// TwinCAT 3 PLC project PLC
// ProgramVersion: 3.1.4023.0
// libraries:
//   EfficientIO Communicator, * (EfficientIO)
//   Lynus Energy Basic, * (Lynus AG)
//   Lynus Energy ModbusRTU, * (Lynus AG)
//   Lynus Energy ModbusTCP, * (Lynus AG)
//   Lynus Persistent Data V1, * (Lynus AG)
//   Lynus Sensor Basic, * (Lynus AG)
//   Lynus Standards, * (Lynus AG)
//   Tc2_ModbusSrv, * (Beckhoff Automation GmbH)
//   Tc2_Standard, * (Beckhoff Automation GmbH)
//   Tc2_System, * (Beckhoff Automation GmbH)
//   Tc2_Utilities, * (Beckhoff Automation GmbH)
//   Tc3_Module, * (Beckhoff Automation GmbH)
// project tree:
//   DUTs/ eByteOrder.TcDUT
//   / Fast_Task.TcTTO, Middle_Task.TcTTO, Slow_Task.TcTTO
//   FBs/ FB_CV_WORD_TO_DWORD.TcPOU, FB_EnergyCounter.TcPOU, FB_Honeywell_Excange_Data.TcPOU, FB_HouseC_Power_Virtual_v2.TcPOU
//   POUs/ prgComLynus.TcPOU, prgCS.TcPOU, prgEHE.TcPOU, prgEMS.TcPOU, prgGrid.TcPOU, prgHoneywell.TcPOU, prgHouse.TcPOU, prgKNX.TcPOU, prgPerData.TcPOU, prgPV.TcPOU, prgRWLynus.TcPOU, prgVarLynus.TcPOU, prgXelect.TcPOU
// real-time tasks:
//   TASK Fast Task: cycle T#5ms, priority 6, ADS port 351
//   TASK Middle Task: cycle T#10ms, priority 8, ADS port 352
//   TASK Slow Task: cycle T#20ms, priority 10, ADS port 353
// I/O:
//   DEVICE Gerät 2 (CX-BK)
//     Box 1 (CX-BK)
// variable links:
//   PLC/PLC Instance <-> Device 2 (CX-BK)/Box 1 (CX-BK)
//     Fast_Task Inputs/prgCS.fbRTUMaster.fbmodbusmaster.InData/D[{0..21}] <-> Term 4 (KL6041)/Channel 1/Data In {0..21}  (22 links)
//     Fast_Task Inputs/prgCS.fbRTUMaster.fbmodbusmaster.InData/Status <-> Term 4 (KL6041)/Channel 1/Status
//     Fast_Task Inputs/prgKNX.fbKBusState.uiKBusState_OUT <-> Inputs/State
//     Fast_Task Outputs/prgCS.fbRTUMaster.fbmodbusmaster.OutData/Ctrl <-> Term 4 (KL6041)/Channel 1/Ctrl
//     Fast_Task Outputs/prgCS.fbRTUMaster.fbmodbusmaster.OutData/D[{0..21}] <-> Term 4 (KL6041)/Channel 1/Data Out {0..21}  (22 links)
//     Middle_Task Inputs/prgEHE.fbH08_1.fbAOEHE.usiState <-> Term 2 (KL4404)/Channel 1/Status
//     Middle_Task Inputs/prgEHE.fbH08_2.fbAOEHE.usiState <-> Term 2 (KL4404)/Channel 2/Status
//     Middle_Task Inputs/prgEHE.fbH09_1.fbAOEHE.usiState <-> Term 2 (KL4404)/Channel 3/Status
//     Middle_Task Inputs/prgKNX.fbKNXMaster.arrKNXKL6301ComIn @bit {16..184 step 8} <-> Term 3 (KL6301)/Channel 1/Input Data {1..22}  (22 links)
//     Middle_Task Inputs/prgKNX.fbKNXMaster.arrKNXKL6301ComIn <-> Term 3 (KL6301)/Channel 1/Parameter Status
//     Middle_Task Outputs/prgEHE.fbH08_1.fbAOEHE.iDataOut <-> Term 2 (KL4404)/Channel 1/Daten Aus
//     Middle_Task Outputs/prgEHE.fbH08_2.fbAOEHE.iDataOut <-> Term 2 (KL4404)/Channel 2/Daten Aus
//     Middle_Task Outputs/prgEHE.fbH09_1.fbAOEHE.iDataOut <-> Term 2 (KL4404)/Channel 3/Daten Aus
//     Middle_Task Outputs/prgKNX.fbKNXMaster.arrKNXKL6301ComOut @bit {16..184 step 8} <-> Term 3 (KL6301)/Channel 1/Output Data {1..22}  (22 links)
//     Middle_Task Outputs/prgKNX.fbKNXMaster.arrKNXKL6301ComOut <-> Term 3 (KL6301)/Channel 1/Parameter Control

CONFIGURATION PLC
    RESOURCE PLC ON TwinCAT3
        TASK Fast_Task(INTERVAL := T#5ms, PRIORITY := 6);
        TASK Middle_Task(INTERVAL := T#10ms, PRIORITY := 8);
        TASK Slow_Task(INTERVAL := T#20ms, PRIORITY := 10);
        PROGRAM prgRWLynus WITH Fast_Task : prgRWLynus;
        PROGRAM prgVarLynus WITH Fast_Task : prgVarLynus;
        PROGRAM prgCS WITH Fast_Task : prgCS;
        PROGRAM prgEHE WITH Middle_Task : prgEHE;
        PROGRAM prgEMS WITH Middle_Task : prgEMS;
        PROGRAM prgHoneywell WITH Middle_Task : prgHoneywell;
        PROGRAM prgKNX WITH Middle_Task : prgKNX;
        PROGRAM prgPV WITH Middle_Task : prgPV;
        PROGRAM prgXelect WITH Middle_Task : prgXelect;
        PROGRAM prgPerData WITH Middle_Task : prgPerData;
        PROGRAM prgHouse WITH Middle_Task : prgHouse;
        PROGRAM prgGrid WITH Middle_Task : prgGrid;
        PROGRAM prgComLynus WITH Slow_Task : prgComLynus;
    END_RESOURCE
END_CONFIGURATION

// ---- DUTs/eByteOrder.TcDUT
TYPE eByteOrder :
(
	eBigEndian	:= 0,
	eLittleEndian	:= 1
);
END_TYPE

// ---- POUs/prgRWLynus.TcPOU
PROGRAM prgRWLynus
VAR
	fbRW1		: FB_ReadWrite;
	fbRW2		: FB_ReadWrite;
	fbRW3		: FB_ReadWrite;
	fbRW4		: FB_ReadWrite;
	fbRW5		: FB_ReadWrite;
	fbRW6		: FB_ReadWrite;
END_VAR

fbRW1();
fbRW2();
fbRW3();
fbRW4();
fbRW5();
fbRW6();

END_PROGRAM

// ---- POUs/prgVarLynus.TcPOU
PROGRAM prgVarLynus
VAR
	fbVar			: FB_VarInfo;
END_VAR

fbVar(
	bReadInfo:= , 
	eTMCFile:= eSelectTMCFile.eUseTMCFile, 
	eSavePositionTMCFile:= eSavePositionOnPLC.ePostionHardDisk, 
	udiCounterFoundVariables=> , 
	bError=> , 
	bBusy=> , 
	byProgress=> , 
	udiErrorCodeOut=> , 
	eErrorVarInfo_Out=> , 
	sVarWithError=> );

END_PROGRAM

// ---- POUs/prgCS.TcPOU
PROGRAM prgCS
VAR
	fbRTUMaster					: FB_KL6xxx_ModbusRTU_22B_Master;
	byErrorwarningRTU			: BYTE;									//{#lynus.ag#()}
	fbCS1						: FB_ECS_Schrack_EM_CionHome;			//{#lynus.ag#()}
	fbCS2						: FB_ECS_Schrack_EM_CionHome;			//{#lynus.ag#()}
	fbCS3						: FB_ECS_Schrack_EM_CionHome;			//{#lynus.ag#()}
	bCarConnCS1					: BOOL;									//{#lynus.ag#()}
	bCarConnCS2					: BOOL;									//{#lynus.ag#()}
	bCarConnCS3					: BOOL;									//{#lynus.ag#()}
	bOnEmergPowerOffCS1			: BOOL;									//{#lynus.ag#()}
	bOnEmergPowerOffCS2			: BOOL;									//{#lynus.ag#()}
	bOnEmergPowerOffCS3			: BOOL;									//{#lynus.ag#()}
	bSOnEmergPowerOffCS1		: BOOL;									//{#lynus.ag#()}
	bSOnEmergPowerOffCS2		: BOOL;									//{#lynus.ag#()}
	bSOnEmergPowerOffCS3		: BOOL;									//{#lynus.ag#()}
	byErrorWarningCS1			: BYTE;									//{#lynus.ag#()}
	byErrorWarningCS2			: BYTE;									//{#lynus.ag#()}
	byErrorWarningCS3			: BYTE;									//{#lynus.ag#()}
	wCPStateCS1					: WORD;									//{#lynus.ag#()}
	bChargingReleaseInavlidCS1	: BOOL;									//{#lynus.ag#()}
	rChargingTimeInMinCS1		: REAL;									//{#lynus.ag#()}
	wCPStateCS2					: WORD;									//{#lynus.ag#()}
	bChargingReleaseInavlidCS2	: BOOL;									//{#lynus.ag#()}
	rChargingTimeInMinCS2		: REAL;									//{#lynus.ag#()}
	wCPStateCS3					: WORD;									//{#lynus.ag#()}
	bChargingReleaseInavlidCS3	: BOOL;									//{#lynus.ag#()}
	rChargingTimeInMinCS3		: REAL;									//{#lynus.ag#()}
	byErrorCounter				: BYTE;									//{#lynus.ag#()}
	FpErrror					: R_TRIG;
END_VAR

//Power Data
//Each CS has 14kW

fbRTUMaster(
	bConfigTerminal:= , 
	uiKBusState_IN:= prgKNX.fbKBusState.uiKBusState_OUT, 
	bBusy=> , 
	byErrorWarning=> , 
	byActualAdressInUse=> , 
	diNrOfMBRTUMasterLine_OUT=> , 
	eMessageMBRTUMaster=> , 
	bTerminalIsConfigured=> );

fbRTUMaster(
	bConfigTerminal:= , 
	bBusy=> , 
	byErrorWarning=> , 
	diNrOfMBRTUMasterLine_OUT=> , 
	eMessageMBRTUMaster=> , 
	bTerminalIsConfigured=> );

byErrorwarningRTU := fbRTUMaster.byErrorWarning;

FpErrror(CLK:= byErrorwarningRTU = 2, Q=> );
	IF FpErrror.Q THEN byErrorCounter := byErrorCounter + 1; END_IF
	
//Garage 1 near Door	
fbCS1.stSetupECS.bOnEmergPowerOff := bOnEmergPowerOffCS1;

fbCS1(
	bEnable:= , 
	bPowerDataInvers:= , 
	byMBAdress:= 1, 
	diNrOfMBRTUMasterLine_IN:= fbRTUMaster.diNrOfMBRTUMasterLine_OUT, 
	diNrOfEMS_IN:= prgEMS.EMS.diNrOfEMS_OUT, 
	diNrOfEM_IN_CS:= , 
	stSetupECS:= , 
	stDataECS=> , 
	eSchrackErrors=> , 
	diNrOfECS_OUT=> );

wCPStateCS1:= fbCS1.wCPStateECS;
	bChargingReleaseInavlidCS1 := fbCS1.bChargingReleaseInavlid;
		rChargingTimeInMinCS1 := fbCS1.stDataECS.arrChargingTimeInMin[1];
			byErrorWarningCS1 := fbCS1.stDataECS.byErrorWarning;
				bCarConnCS1 := fbCS1.stDataECS.bCarConnected;
					bSOnEmergPowerOffCS1 := fbCS1.stDataECS.bSOnEmergPowerOff;
	
//Between CS1	
fbCS2.stSetupECS.bOnEmergPowerOff := bOnEmergPowerOffCS2;

fbCS2(
	bEnable:= , 
	bPowerDataInvers:= , 
	byMBAdress:= 2, 
	diNrOfMBRTUMasterLine_IN:= fbRTUMaster.diNrOfMBRTUMasterLine_OUT, 
	diNrOfEMS_IN:= prgEMS.EMS.diNrOfEMS_OUT, 
	diNrOfEM_IN_CS:= , 
	stSetupECS:= , 
	stDataECS=> , 
	eSchrackErrors=> , 
	diNrOfECS_OUT=> );

wCPStateCS2:= fbCS2.wCPStateECS;
	bChargingReleaseInavlidCS2 := fbCS2.bChargingReleaseInavlid;
		rChargingTimeInMinCS2 := fbCS2.stDataECS.arrChargingTimeInMin[1];
			byErrorWarningCS2 := fbCS2.stDataECS.byErrorWarning;
				bCarConnCS2 := fbCS2.stDataECS.bCarConnected;
					bSOnEmergPowerOffCS2 := fbCS2.stDataECS.bSOnEmergPowerOff;	
	
//Outdoor CS
fbCS3.stSetupECS.bOnEmergPowerOff := bOnEmergPowerOffCS3;

fbCS3(
	bEnable:= , 
	bPowerDataInvers:= , 
	byMBAdress:= 3, 
	diNrOfMBRTUMasterLine_IN:= fbRTUMaster.diNrOfMBRTUMasterLine_OUT, 
	diNrOfEMS_IN:= prgEMS.EMS.diNrOfEMS_OUT, 
	diNrOfEM_IN_CS:= , 
	stSetupECS:= , 
	stDataECS=> , 
	eSchrackErrors=> , 
	diNrOfECS_OUT=> );
	
wCPStateCS3:= fbCS3.wCPStateECS;
	bChargingReleaseInavlidCS3 := fbCS3.bChargingReleaseInavlid;
		rChargingTimeInMinCS3 := fbCS3.stDataECS.arrChargingTimeInMin[1];
			byErrorWarningCS3 := fbCS3.stDataECS.byErrorWarning;
				bCarConnCS3 := fbCS3.stDataECS.bCarConnected;
					bSOnEmergPowerOffCS3 := fbCS3.stDataECS.bSOnEmergPowerOff;

END_PROGRAM

// ---- POUs/prgKNX.TcPOU
PROGRAM prgKNX
VAR
	fbKBusState				: FB_K_Bus_State;
	fbKNXMaster				: FB_KL6301_KNX_Master;
	fbRampHeating			: FB_OBC_OnOff_KNX;				//{#lynus.ag#()}
	fbTreeHeating			: FB_OBC_OnOff_KNX;				//{#lynus.ag#()}
	fbPumpFishSea			: FB_OBC_OnOff_KNX;				//{#lynus.ag#()}
	fbPumpSwimSea			: FB_OBC_OnOff_KNX;				//{#lynus.ag#()}
	bOnEmergPowerOffRH		: BOOL;							//{#lynus.ag#()}
	bOnEmergPowerOffTH		: BOOL;							//{#lynus.ag#()}
	bOnEmergPowerOffPFish	: BOOL;							//{#lynus.ag#()}
	bOnEmergPowerOffPSwim	: BOOL;							//{#lynus.ag#()}
	bSOnEmergPowerOffRH		: BOOL;							//{#lynus.ag#()}
	bSOnEmergPowerOffTH		: BOOL;							//{#lynus.ag#()}
	bSOnEmergPowerOffPFish	: BOOL;							//{#lynus.ag#()}
	bSOnEmergPowerOffPSwim	: BOOL;							//{#lynus.ag#()}
	byErrorWarningRH		: BYTE;							//{#lynus.ag#()}
	byErrorWarningTH		: BYTE;							//{#lynus.ag#()}
	byErrorWarningPFish		: BYTE;							//{#lynus.ag#()}
	byErrorWarningPSwim		: BYTE;							//{#lynus.ag#()}
END_VAR

//Power Data
//Ramp Heating 34kw
//Three Heating 13kW 
//Fish Sea pump 7.5kW
//Swim Sea Pump 7.5kw

//K-Bus State
fbKBusState(uiKBusState_OUT=> );

//Configure the KXN Master
fbKNXMaster.stPhysAddrTerminal.Area := 1;
	fbKNXMaster.stPhysAddrTerminal.Device := 160;
		fbKNXMaster.stPhysAddrTerminal.Line := 9;
		
fbKNXMaster.arrGroupFilter[1].GROUP_ADDR.MAIN := 6;
	fbKNXMaster.arrGroupFilter[1].GROUP_ADDR.NUMBER := 0;
		fbKNXMaster.arrGroupFilter[1].GROUP_ADDR.SUB_MAIN := 1;
fbKNXMaster.arrGroupFilter[1].GROUP_LEN := 4;	
	
fbKNXMaster(
	stPhysAddrTerminal:= , 
	arrGroupFilter:= , 
	iKL6301Mode:= 0, 
	uiKBusState_IN:= fbKBusState.uiKBusState_OUT, 
	bActive=> , 
	bReady=> , 
	byErrorWarning=> , 
	diNrOfKNXMasterLine_OUT=> , 
	eMessageKNXMaster=> );

fbTreeHeating.strGroupAddr.MAIN := 6;
	fbTreeHeating.strGroupAddr.SUB_MAIN := 1;
		fbTreeHeating.strGroupAddr.NUMBER := 0;	

fbTreeHeating.stSetupOBC.bOnEmergPowerOff := bOnEmergPowerOffTH;
	
fbTreeHeating(
	bEnable:= , 
	bPowerDataInvers:= , 
	diNrOfKNXMasterLine_IN:= fbKNXMaster.diNrOfKNXMasterLine_OUT, 
	diNrOfEMS_IN:= prgEMS.EMS.diNrOfEMS_OUT, 
	diNrOfEM_IN_OBC:= , 
	stSetupOBC:= , 
	strGroupAddr:= , 
	stDataOBC=> , 
	diNrOfOBC_OUT=> );

byErrorWarningTH := fbTreeHeating.stDataOBC.byErrorWarning;	
	bSOnEmergPowerOffTH := fbTreeHeating.stDataOBC.bSOnEmergPowerOff;	
	
fbPumpFishSea.strGroupAddr.MAIN := 6;
	fbPumpFishSea.strGroupAddr.SUB_MAIN := 1;
		fbPumpFishSea.strGroupAddr.NUMBER := 2;	

fbPumpFishSea.stSetupOBC.bOnEmergPowerOff := bOnEmergPowerOffPFish;
	
fbPumpFishSea(
	bEnable:= , 
	bPowerDataInvers:= , 
	diNrOfKNXMasterLine_IN:= fbKNXMaster.diNrOfKNXMasterLine_OUT, 
	diNrOfEMS_IN:= prgEMS.EMS.diNrOfEMS_OUT, 
	diNrOfEM_IN_OBC:= , 
	stSetupOBC:= , 
	strGroupAddr:= , 
	stDataOBC=> , 
	diNrOfOBC_OUT=> );

byErrorWarningPFish := fbPumpFishSea.stDataOBC.byErrorWarning;
	bSOnEmergPowerOffPFish := fbPumpFishSea.stDataOBC.bSOnEmergPowerOff;		
	
fbPumpSwimSea.strGroupAddr.MAIN := 6;
	fbPumpSwimSea.strGroupAddr.SUB_MAIN := 1;
		fbPumpSwimSea.strGroupAddr.NUMBER := 3;	

fbPumpSwimSea.stSetupOBC.bOnEmergPowerOff := bOnEmergPowerOffPSwim;
	
fbPumpSwimSea(
	bEnable:= , 
	bPowerDataInvers:= , 
	diNrOfKNXMasterLine_IN:= fbKNXMaster.diNrOfKNXMasterLine_OUT, 
	diNrOfEMS_IN:= prgEMS.EMS.diNrOfEMS_OUT, 
	diNrOfEM_IN_OBC:= , 
	stSetupOBC:= , 
	strGroupAddr:= , 
	stDataOBC=> , 
	diNrOfOBC_OUT=> );

byErrorWarningPSwim := fbPumpSwimSea.stDataOBC.byErrorWarning;	
	bSOnEmergPowerOffPSwim := fbPumpSwimSea.stDataOBC.bSOnEmergPowerOff;
	
fbRampHeating.strGroupAddr.MAIN := 6;
	fbRampHeating.strGroupAddr.SUB_MAIN := 1;
		fbRampHeating.strGroupAddr.NUMBER := 1;	

fbRampHeating.stSetupOBC.bOnEmergPowerOff := bOnEmergPowerOffRH;
	
fbRampHeating(
	bEnable:= , 
	bPowerDataInvers:= , 
	diNrOfKNXMasterLine_IN:= fbKNXMaster.diNrOfKNXMasterLine_OUT, 
	diNrOfEMS_IN:= prgEMS.EMS.diNrOfEMS_OUT, 
	diNrOfEM_IN_OBC:= , 
	stSetupOBC:= , 
	strGroupAddr:= , 
	stDataOBC=> , 
	diNrOfOBC_OUT=> );
	
byErrorWarningRH := fbRampHeating.stDataOBC.byErrorWarning;	
	bSOnEmergPowerOffRH := fbRampHeating.stDataOBC.bSOnEmergPowerOff;

END_PROGRAM

// ---- POUs/prgEMS.TcPOU
PROGRAM prgEMS
VAR
	EMS					: FB_EMS;			//{#lynus.ag#()}
	iMassageEMS			: INT;				//{#lynus.ag#()}
	fbreboot			: NT_Reboot;
END_VAR

EMS(
	bEnable:= , 
	diNrOfEM_IN_ECS:= , 
	stSetupEMS:= , 
	eOperationMode:= ,
	eSpeedModeBackendController:= E_SpeedModeBackendController_EMS.eSlow, 
	eSpeedModeLocalController:= E_SpeedModeLocalController_EMS.eBalanced,
	eMessageEMS=> , 
	bStateEnable=> , 
	bStateAllowChrgFromGrid=> , 
	bMissingPowerData=> , 
	bSurplusAvailable=> , 
	bActivateHP=> , 
	bControllingState=> , 
	byProgress=> , 
	diNrOfEMS_OUT=> , 
	rHeartbeat=> , 
	rErrorWarning=> , 
	rEnergyOptReady=> , 
	rNewBattPower=> , 
	arrMinPrioReached=> , 
	arrMaxPrioReached=> );
	
iMassageEMS := ems.eMessageEMS;

fbreboot(
	NETID:= , 
	DELAY:= , 
	START:= , 
	TMOUT:= , 
	BUSY=> , 
	ERR=> , 
	ERRID=> );

END_PROGRAM

// ---- POUs/prgEHE.TcPOU
PROGRAM prgEHE
VAR
	fbTempH08					: FB_TempS_Ext_Input;
	fbTempH09					: FB_TempS_Ext_Input;
	fbH08_1						: FB_EHE_Linear_AO;			//{#lynus.ag#()}
	fbH08_2						: FB_EHE_Linear_AO;			//{#lynus.ag#()}
	fbH09_1						: FB_EHE_Linear_AO;			//{#lynus.ag#()}
	bSOnEmergPowerOffH08_1		: BOOL;						//{#lynus.ag#()}
	bSOnEmergPowerOffH08_2		: BOOL;						//{#lynus.ag#()}
	bSOnEmergPowerOffH09_1		: BOOL;						//{#lynus.ag#()}
	byErrorWarningH08_1			: BYTE;						//{#lynus.ag#()}
	byErrorWarningH08_2			: BYTE;						//{#lynus.ag#()}
	byErrorWarningH09_1			: BYTE;						//{#lynus.ag#()}
END_VAR
VAR PERSISTENT
	bOnEmergPowerOffH08_1		: BOOL;						//{#lynus.ag#()}
	bOnEmergPowerOffH08_2		: BOOL;						//{#lynus.ag#()}
	bOnEmergPowerOffH09_1		: BOOL;						//{#lynus.ag#()}
END_VAR

//Power Data
//each Heating Element 9kW

fbTempH08(
	bEnable:= TRUE, 
	rTemperatureOffset:= , 
	bExtErrorTemp:= prgHoneywell.fbHoneywellCntr.bErrorFunction OR prgHoneywell.fbHoneywellCntr.bErrorTemp_H08_Below OR prgHoneywell.fbHoneywellCntr.bErrorTemp_H08_Top, 
	rExtTempValue:= (prgHoneywell.fbHoneywellCntr.rBufferTemp_H08_Below + prgHoneywell.fbHoneywellCntr.rBufferTemp_H08_Top) / 2, 
	stDataTempS=> , 
	diNrOfTempS_OUT=> );
	
fbTempH09(
	bEnable:= TRUE, 
	rTemperatureOffset:= , 
	bExtErrorTemp:= prgHoneywell.fbHoneywellCntr.bErrorFunction OR prgHoneywell.fbHoneywellCntr.bErrorTemp_H09_WW, 
	rExtTempValue:= prgHoneywell.fbHoneywellCntr.rBufferTemp_H09_WW, 
	stDataTempS=> , 
	diNrOfTempS_OUT=> );

//Buffer House	
fbH08_1.stSetupEHE.bOnEmergPowerOff := bOnEmergPowerOffH08_1;
	fbH08_1.stSetupEHE.bDisableLegionellaPr := TRUE;
	
fbH08_1(
	bEnable:= , 
	bPowerDataInvers:= , 
	bNoLinear:= FALSE,
	diNrOfEMS_IN:= prgEMS.EMS.diNrOfEMS_OUT, 
	diNrOfEM_IN_EHE:= , 
	diNrOfTempS_IN:= fbTempH08.diNrOfTempS_OUT, 
	stSetupEHE:= , 
	stDataEHE=> , 
	diNrOfEHE_OUT=> , 
	rTargetPowerForExtFunc=> );	
	
byErrorWarningH08_1 := fbH08_1.stDataEHE.byErrorWarning;
	bSOnEmergPowerOffH08_1 := fbH08_1.stDataEHE.bSOnEmergPowerOff;

fbH08_2.stSetupEHE.bOnEmergPowerOff := bOnEmergPowerOffH08_2;
	fbH08_2.stSetupEHE.bDisableLegionellaPr := TRUE;
	
fbH08_2(
	bEnable:= , 
	bPowerDataInvers:= , 
	bNoLinear:= FALSE,
	diNrOfEMS_IN:= prgEMS.EMS.diNrOfEMS_OUT, 
	diNrOfEM_IN_EHE:= , 
	diNrOfTempS_IN:= fbTempH08.diNrOfTempS_OUT, 
	stSetupEHE:= , 
	stDataEHE=> , 
	diNrOfEHE_OUT=> , 
	rTargetPowerForExtFunc=> );

byErrorWarningH08_2 := fbH08_2.stDataEHE.byErrorWarning;
	bSOnEmergPowerOffH08_2 := fbH08_2.stDataEHE.bSOnEmergPowerOff;	
	
//Warmwater Boiler	
fbH09_1.stSetupEHE.bOnEmergPowerOff := bOnEmergPowerOffH09_1;

fbH09_1(
	bEnable:= , 
	bPowerDataInvers:= , 
	bNoLinear:= FALSE,
	diNrOfEMS_IN:= prgEMS.EMS.diNrOfEMS_OUT, 
	diNrOfEM_IN_EHE:= , 
	diNrOfTempS_IN:= fbTempH09.diNrOfTempS_OUT, 
	stSetupEHE:= , 
	stDataEHE=> , 
	diNrOfEHE_OUT=> , 
	rTargetPowerForExtFunc=> );
	
byErrorWarningH09_1 := fbH09_1.stDataEHE.byErrorWarning;
	bSOnEmergPowerOffH09_1 := fbH09_1.stDataEHE.bSOnEmergPowerOff;

END_PROGRAM

// ---- POUs/prgHoneywell.TcPOU
PROGRAM prgHoneywell
VAR
	fbHoneywellCntr			: FB_Honeywell_Excange_Data;
	fbTempH01				: FB_TempS_Ext_Input;
	fbH01_1					: FB_EHE_Linear_AO;			//{#lynus.ag#()}
	fbH01_2					: FB_EHE_Linear_AO;			//{#lynus.ag#()}
	fbH01_3					: FB_EHE_Linear_AO;			//{#lynus.ag#()}
	bSOnEmergPowerOffH01_1	: BOOL;						//{#lynus.ag#()}
	bSOnEmergPowerOffH01_2	: BOOL;						//{#lynus.ag#()}
	bSOnEmergPowerOffH01_3	: BOOL;						//{#lynus.ag#()}
	rBufferTemp_H01_Top		: REAL;						//{#lynus.ag#()}
	rBufferTemp_H01_Below	: REAL;						//{#lynus.ag#()}
	rBufferTemp_H08_Top		: REAL;						//{#lynus.ag#()}
	rBufferTemp_H08_Below	: REAL;						//{#lynus.ag#()}
	bErrorHoneywell			: BOOL;						//{#lynus.ag#()}
	byErrorWarningH01_1		: BYTE;						//{#lynus.ag#()}
	byErrorWarningH01_2		: BYTE;						//{#lynus.ag#()}
	byErrorWarningH01_3		: BYTE;						//{#lynus.ag#()}
	dwHeatingMeterHouse		: DWORD;					//{#lynus.ag#()}
	dwHeatingMeterStable	: DWORD;					//{#lynus.ag#()}
	dwWaterMeterMain1		: DWORD;					//{#lynus.ag#()}
	dwWaterMeterService1	: DWORD;					//{#lynus.ag#()}
	dwWaterMeterStable1		: DWORD;					//{#lynus.ag#()}
	dwElectricMeterCounter	: DWORD;					//{#lynus.ag#()}
	dwElectricMeterPower	: LREAL;					//{#lynus.ag#()}
END_VAR
VAR PERSISTENT
	bOnEmergPowerOffH01_1	: BOOL;						//{#lynus.ag#()}
	bOnEmergPowerOffH01_2	: BOOL;						//{#lynus.ag#()}
	bOnEmergPowerOffH01_3	: BOOL;						//{#lynus.ag#()}
END_VAR

//Creator : Kai Ebensperger
//Company : Lynus AG
//Updated : M.Schwarzmann
//Date : 11.07.2022
//Version : 1.0.0.4

//changes
//1.0.0.1 : added dwWaterMeterMain, dwWaterMeterService, dwElectricMeterCounter, dwElectricMeterPower at fbHoneywellCntr
//1.0.0.2 : changed Variable dwElectricMeterPower from Type REAL to LREAL
//1.0.0.3 : re-named Variables dwWaterMeterMain, dwWaterMeterService
//1.0.0.4 : added dwWaterMeterStable1


//Power Data
//Each EHE 9 kW

fbHoneywellCntr(
	bEnable:= TRUE, 
	byUnitID:= 1, 
	rTargetPowerEHEH01_1:= fbH01_1.rTargetPowerForExtFunc, 
	rTargetPowerEHEH01_2:= fbH01_2.rTargetPowerForExtFunc, 
	rTargetPowerEHEH01_3:= fbH01_3.rTargetPowerForExtFunc, 
	rTargetPowerEHEH08_1:= prgEHE.fbH08_1.rTargetPowerForExtFunc, 
	rTargetPowerEHEH08_2:= prgEHE.fbH08_2.rTargetPowerForExtFunc, 
	rTargetPowerEHEH09_1:= prgEHE.fbH09_1.rTargetPowerForExtFunc, 
	sIPAdress:= '10.68.10.60', 
	bErrorTemp_H01_Top=> , 
	bErrorTemp_H01_Below=> , 
	bErrorTemp_H08_Top=> , 
	bErrorTemp_H08_Below=> , 
	bErrorTemp_H09_WW=> , 
	bErrorFunction=> bErrorHoneywell, 
	dwHeatingMeterHouse=> dwHeatingMeterHouse,
	dwHeatingMeterStable=> dwHeatingMeterStable,
	dwWaterMeterMain1=> dwWaterMeterMain1,
	dwWaterMeterService1=> dwWaterMeterService1,
	dwWaterMeterStable1=> dwWaterMeterStable1,
	dwElectricMeterCounter=> dwElectricMeterCounter,
	dwElectricMeterPower=> dwElectricMeterPower,
	rBufferTemp_H01_Top=> rBufferTemp_H01_Top, 
	rBufferTemp_H01_Below=> rBufferTemp_H01_Below, 
	rBufferTemp_H08_Top=> rBufferTemp_H08_Top, 
	rBufferTemp_H08_Below=> rBufferTemp_H08_Below, 
	rBufferTemp_H09_WW=> );

fbTempH01(
	bEnable:= TRUE, 
	rTemperatureOffset:= , 
	bExtErrorTemp:= fbHoneywellCntr.bErrorFunction OR fbHoneywellCntr.bErrorTemp_H01_Below OR fbHoneywellCntr.bErrorTemp_H01_Top, 
	rExtTempValue:= (fbHoneywellCntr.rBufferTemp_H01_Below + fbHoneywellCntr.rBufferTemp_H01_Top) / 2, 
	stDataTempS=> , 
	diNrOfTempS_OUT=> );

//Buffer Workshop 	
fbH01_1.stSetupEHE.bOnEmergPowerOff := bOnEmergPowerOffH01_1;
	fbH01_1.stSetupEHE.bDisableLegionellaPr := TRUE;
	
fbH01_1(
	bEnable:= , 
	bPowerDataInvers:= , 
	bNoLinear:= FALSE,
	diNrOfEMS_IN:= prgEMS.EMS.diNrOfEMS_OUT, 
	diNrOfEM_IN_EHE:= , 
	diNrOfTempS_IN:= fbTempH01.diNrOfTempS_OUT, 
	stSetupEHE:= , 
	stDataEHE=> , 
	diNrOfEHE_OUT=> , 
	rTargetPowerForExtFunc=> );

byErrorWarningH01_1 := fbH01_1.stDataEHE.byErrorWarning;
	bSOnEmergPowerOffH01_1 := fbH01_1.stDataEHE.bSOnEmergPowerOff;	

fbH01_2.stSetupEHE.bOnEmergPowerOff := bOnEmergPowerOffH01_2;
	fbH01_2.stSetupEHE.bDisableLegionellaPr := TRUE;
	
fbH01_2(
	bEnable:= , 
	bPowerDataInvers:= , 
	bNoLinear:= FALSE,
	diNrOfEMS_IN:= prgEMS.EMS.diNrOfEMS_OUT, 
	diNrOfEM_IN_EHE:= , 
	diNrOfTempS_IN:= fbTempH01.diNrOfTempS_OUT, 
	stSetupEHE:= , 
	stDataEHE=> , 
	diNrOfEHE_OUT=> , 
	rTargetPowerForExtFunc=> );

byErrorWarningH01_2 := fbH01_2.stDataEHE.byErrorWarning;
	bSOnEmergPowerOffH01_2 := fbH01_2.stDataEHE.bSOnEmergPowerOff;	

fbH01_3.stSetupEHE.bOnEmergPowerOff := bOnEmergPowerOffH01_3;
	fbH01_3.stSetupEHE.bDisableLegionellaPr := TRUE;
	
fbH01_3(
	bEnable:= , 
	bPowerDataInvers:= , 
	bNoLinear:= FALSE,
	diNrOfEMS_IN:= prgEMS.EMS.diNrOfEMS_OUT, 
	diNrOfEM_IN_EHE:= , 
	diNrOfTempS_IN:= fbTempH01.diNrOfTempS_OUT, 
	stSetupEHE:= , 
	stDataEHE=> , 
	diNrOfEHE_OUT=> , 
	rTargetPowerForExtFunc=> );
	
byErrorWarningH01_3 := fbH01_3.stDataEHE.byErrorWarning;
	bSOnEmergPowerOffH01_3 := fbH01_3.stDataEHE.bSOnEmergPowerOff;

END_PROGRAM

// ---- FBs/FB_Honeywell_Excange_Data.TcPOU
FUNCTION_BLOCK FB_Honeywell_Excange_Data
VAR_INPUT
	bEnable							: BOOL;					//Enable the Function
	byUnitID						: BYTE;					//Unit ID fromt the Honeywell controller (0 to 255)		
	rTargetPowerEHEH01_1			: REAL;					//Target power for the EHE H01_1 to send to the Honeywell controller (Scalefactor is * 10) 										
	rTargetPowerEHEH01_2			: REAL;					//Target power for the EHE H01_2 to send to the Honeywell controller (Scalefactor is * 10)
	rTargetPowerEHEH01_3			: REAL;					//Target power for the EHE H01_3 to send to the Honeywell controller (Scalefactor is * 10)
	rTargetPowerEHEH08_1			: REAL;					//Target power for the EHE H08_1 to send to the Honeywell controller (Only to show on the internal house visualization) (Scalefactor is * 10)
	rTargetPowerEHEH08_2			: REAL;					//Target power for the EHE H08_2 to send to the Honeywell controller (Only to show on the internal house visualization) (Scalefactor is * 10)
	rTargetPowerEHEH09_1			: REAL;					//Target power for the EHE H09_1 to send to the Honeywell controller (Only to show on the internal house visualization) (Scalefactor is * 10)
	sIPAdress						: STRING(15);			//IP Adress from the Honeywell controller
END_VAR
VAR_OUTPUT
	bErrorTemp_H01_Top				: BOOL;					//True, when this Temp. senor has a error 
	bErrorTemp_H01_Below			: BOOL;					//True, when this Temp. senor has a error 
	bErrorTemp_H08_Top				: BOOL;					//True, when this Temp. senor has a error 
	bErrorTemp_H08_Below			: BOOL;					//True, when this Temp. senor has a error 
	bErrorTemp_H09_WW				: BOOL;					//True, when this Temp. senor has a error 
	bErrorFunction					: BOOL;					//Modbus TCP Error or Timout Error
	dwHeatingMeterHouse				: DWORD;				//Heating Meter value House in kWh
	dwHeatingMeterStable			: DWORD;				//Heating Meter value Stable in kWh
	rBufferTemp_H01_Top				: REAL;					//Temp. Value from this sensor (Scalfactor is / 10)
	rBufferTemp_H01_Below			: REAL;					//Temp. Value from this sensor (Scalfactor is / 10)
	rBufferTemp_H08_Top				: REAL;					//Temp. Value from this sensor (Scalfactor is / 10)
	rBufferTemp_H08_Below			: REAL;					//Temp. Value from this sensor (Scalfactor is / 10)
	rBufferTemp_H09_WW				: REAL;					//Temp. Value from this sensor (Scalfactor is / 10)
	dwWaterMeterMain1				: DWORD;				//Water Meter value Main in m3
	dwWaterMeterService1			: DWORD;				//Water Meter value Service in m3
	dwWaterMeterStable1				: DWORD;				//Water Meter value Service in m3
	dwElectricMeterCounter			: DWORD;				//Electric Meter Counter value in kWh
	dwElectricMeterPowerRaw			: DWORD;				//Electric Meter Power value in W
	dwElectricMeterPower			: LREAL;				//Electric Meter Power value in kW
END_VAR
VAR
	fbMBRead_FC4					: FB_MBReadInputRegs;	//Modbus Read Function (FC4)
	fbMBWrite_FC16					: FB_MBWriteRegs;		//Modbus Write Function (FC16)
	timDelay						: TON;					//Timer for Delay between Request
	timTimeout						: TON;					//Timer for Timeout
	timHB							: TON;					//Timer HB between Lynus and Honeywell
	FPEnable						: R_TRIG;				//Internal positive Edge
	FPError_FC_4					: R_TRIG;				//Internal positive Edge
	FPError_FC_16					: R_TRIG;				//Internal positive Edge
	fbConvert						: FB_CV_WORD_TO_DWORD;	//Convert 2 Word in Dword
	arrBuffer_FC4					: ARRAY[1..14] OF WORD;	//Buffer with Data from FC4
	arrBuffer_FC16					: ARRAY[1..7] OF WORD;	//Buffer with Data from FC16
	byHBCounter						: BYTE;					//HB counter between Lynus and Honeywell.
	iStateModbusRead				: INT;					//State variable for Statemachine
	iStateModbusWrite				: INT;					//State variable for Statemachine
	iStateModbusError				: INT;					//State variable for Statemachine
	iStateModbus_CP					: INT;					//Compare State variable
END_VAR

//Creator : Kai Ebensperger
//Company : Lynus AG
//Updated : M.Schwarzmann
//Date : 11.07.2022
//Version : 1.0.0.5

//With this Functionblock is possible to communicate with the Honeywell Controller via Modbus TCP
//Lynus send the target power for the Electric heating Elements to the Honeywell controller that this can controll it. 
//From the Honeywell Controller we receive the temperature values from each Buffer 
//The Port is 12000 on this project, not modbus typically 502

//changes
//1.0.0.1 : added Water-Meters (Reg: 19, 21), Electric-Meter (Reg: 23, 25)
//1.0.0.2 : added W to kW conversion for dwElectricMeterPower
//1.0.0.3 : changed Variable dwElectricMeterPower from Type REAL to LREAL
//1.0.0.4 : re-named Variables dwWaterMeterMain, dwWaterMeterService
//1.0.0.5 : added Water-Meter (Reg: 27)


(*------------------------------------------------------------------------------------------State Machine Read---------------------------------------------------------------------------------------------*)

//Start the Statemachine
FPEnable(CLK:= bEnable, Q=> );
	IF (FPEnable.Q AND iStateModbusRead = 0 AND iStateModbusRead = 0 AND iStateModbusError = 0) THEN 
		iStateModbusRead := 1; 
	END_IF
		IF NOT bEnable THEN iStateModbusRead := 0; iStateModbusWrite := 0; iStateModbusError := 0; END_IF

//Timer for delay
timDelay(IN:= , PT:= T#250MS, Q=> , ET=> );	

//Timer for Timeout in Statemachine
IF (iStateModbusRead > 0 AND iStateModbusRead <= 4 AND iStateModbusRead = iStateModbus_CP) OR
		(iStateModbusWrite > 0 AND iStateModbusWrite <= 1 AND iStateModbusWrite = iStateModbus_CP) THEN
			timTimeout.IN := TRUE;
ELSE	
			timTimeout.IN := FALSE;
END_IF 
	IF iStateModbusRead = 0 AND iStateModbusWrite = 0 THEN timTimeout.IN := FALSE; END_IF
		timTimeout(IN:= , PT:= T#20S, Q=> , ET=> );

//HB between Lynus and Honeywell
//Switch every Second between 0 and 1
timHB(IN:= NOT timHB.Q, PT:= T#1M, Q=> , ET=> );
	IF timHB.Q THEN byHBCounter := byHBCounter + 1; END_IF
		IF byHBCounter >= 2 THEN byHBCounter := 0; END_IF
		
CASE iStateModbusRead OF
	
	0://Init State
		rBufferTemp_H01_Top := 0;
			rBufferTemp_H01_Below := 0;
				rBufferTemp_H08_Top := 0;
					rBufferTemp_H08_Below := 0;
						rBufferTemp_H09_WW := 0;	

		fbMBRead_FC4.bExecute := FALSE;
			fbMBWrite_FC16.bExecute := FALSE;	
			
	1://Read out all Temperature values
		iStateModbus_CP := iStateModbusRead;
	
		//Reset Write
		fbMBWrite_FC16.bExecute := FALSE;
			arrBuffer_FC16[1] := 0; arrBuffer_FC16[2] := 0; arrBuffer_FC16[3] := 0; arrBuffer_FC16[4] := 0;
					arrBuffer_FC16[5] := 0; arrBuffer_FC16[6] := 0; arrBuffer_FC16[7] := 0;
					
		//Start Read
		fbMBRead_FC4.nQuantity := 5;
			fbMBRead_FC4.nMBAddr := 0;
				fbMBRead_FC4.bExecute := TRUE;	
				
		IF fbMBRead_FC4.bBusy THEN timDelay.IN := TRUE; END_IF
		
		//Wait for Delay, copy Data and then next step
		IF NOT fbMBRead_FC4.bBusy AND NOT fbMBRead_FC4.bError AND timDelay.Q THEN
			//BufferTemp_H01_Top
			rBufferTemp_H01_Top := WORD_TO_REAL(arrBuffer_FC4[1]) / 10; 	
			//BufferTemp_H01_Below
			rBufferTemp_H01_Below := WORD_TO_REAL(arrBuffer_FC4[2]) / 10; 
			//BufferTemp_H08_Top
			rBufferTemp_H08_Top := WORD_TO_REAL(arrBuffer_FC4[3]) / 10;  
			//BufferTemp_H08_Below
			rBufferTemp_H08_Below := WORD_TO_REAL(arrBuffer_FC4[4]) / 10;  
			//BufferTemp_H09_WW
			rBufferTemp_H09_WW := WORD_TO_REAL(arrBuffer_FC4[5]) / 10; 
				//Go to the Next Step
				fbMBRead_FC4.bExecute := FALSE;
					timDelay.IN := FALSE;		
						iStateModbusRead := 2;
		END_IF
			
		//Error or Timeout
		IF FPError_FC_4.Q OR timTimeout.Q THEN
			iStateModbusError := 300;
		END_IF
		
	2://Read out all Temperature states
		iStateModbus_CP := iStateModbusRead;
	
		//Start Read
		fbMBRead_FC4.nQuantity := 5;
			fbMBRead_FC4.nMBAddr := 100;
				fbMBRead_FC4.bExecute := TRUE;	
				
		IF fbMBRead_FC4.bBusy THEN timDelay.IN := TRUE; END_IF
		
		//Wait for Delay, copy Data and then next step
		IF NOT fbMBRead_FC4.bBusy AND NOT fbMBRead_FC4.bError AND timDelay.Q THEN
			//ErrorTemp_H01_Top
			bErrorTemp_H01_Top := WORD_TO_BOOL(arrBuffer_FC4[1]); 	
			//ErrorTemp_H01_Below
			bErrorTemp_H01_Below := WORD_TO_BOOL(arrBuffer_FC4[2]); 
			//ErrorTemp_H08_Top
			bErrorTemp_H08_Top := WORD_TO_BOOL(arrBuffer_FC4[3]);  
			//ErrorTemp_H08_Below
			bErrorTemp_H08_Below := WORD_TO_BOOL(arrBuffer_FC4[4]);  
			//ErrorTemp_H09_WW
			bErrorTemp_H09_WW := WORD_TO_BOOL(arrBuffer_FC4[5]); 
				//Go to the Next Step
				fbMBRead_FC4.bExecute := FALSE;
					timDelay.IN := FALSE;		
						iStateModbusRead := 3;
		END_IF
			
		//Error or Timeout
		IF FPError_FC_4.Q OR timTimeout.Q THEN
			iStateModbusError := 300;
		END_IF
		
	3://Heating Meter Infos House and Stable, Water Meter Infos Main, Service and Stable, Electric Meter with Power
		iStateModbus_CP := iStateModbusRead;
	
		//Start Read
		fbMBRead_FC4.nQuantity := 14;
			fbMBRead_FC4.nMBAddr := 15;
				fbMBRead_FC4.bExecute := TRUE;	
				
		IF fbMBRead_FC4.bBusy THEN timDelay.IN := TRUE; END_IF
		
		//Wait for Delay, copy Data and then next step
		IF NOT fbMBRead_FC4.bBusy AND NOT fbMBRead_FC4.bError AND timDelay.Q THEN
			//Heating Meter Data House
			fbConvert(wInputValue_1:= arrBuffer_FC4[1], wInputValue_2:= arrBuffer_FC4[2], eByteOrderForConvert:= eByteOrder.eBigEndian, dwOutputValue=> dwHeatingMeterHouse);
			//Heating Meter Data Stable
			fbConvert(wInputValue_1:= arrBuffer_FC4[3], wInputValue_2:= arrBuffer_FC4[4], eByteOrderForConvert:= eByteOrder.eBigEndian, dwOutputValue=> dwHeatingMeterStable);
            //Water Meter Data Main-Water
			fbConvert(wInputValue_1:= arrBuffer_FC4[5], wInputValue_2:= arrBuffer_FC4[6], eByteOrderForConvert:= eByteOrder.eBigEndian, dwOutputValue=> dwWaterMeterMain1);
            //Water Meter Data Service-Water
			fbConvert(wInputValue_1:= arrBuffer_FC4[7], wInputValue_2:= arrBuffer_FC4[8], eByteOrderForConvert:= eByteOrder.eBigEndian, dwOutputValue=> dwWaterMeterService1);
            //Electric Meter Data Counter
			fbConvert(wInputValue_1:= arrBuffer_FC4[9], wInputValue_2:= arrBuffer_FC4[10], eByteOrderForConvert:= eByteOrder.eBigEndian, dwOutputValue=> dwElectricMeterCounter);
            //Electric Meter Data Power
			fbConvert(wInputValue_1:= arrBuffer_FC4[11], wInputValue_2:= arrBuffer_FC4[12], eByteOrderForConvert:= eByteOrder.eBigEndian, dwOutputValue=> dwElectricMeterPowerRaw);
			dwElectricMeterPower := DWORD_TO_REAL(dwElectricMeterPowerRaw) / 1000;
			//Water Meter Data Stable-Water
			fbConvert(wInputValue_1:= arrBuffer_FC4[13], wInputValue_2:= arrBuffer_FC4[14], eByteOrderForConvert:= eByteOrder.eBigEndian, dwOutputValue=> dwWaterMeterStable1);	
				//Go to the Next Step
				fbMBRead_FC4.bExecute := FALSE;
					timDelay.IN := FALSE;		
						iStateModbusRead := 4;
		END_IF
			
		//Error or Timeout
		IF FPError_FC_4.Q OR timTimeout.Q THEN
			iStateModbusError := 300;
		END_IF
			
	4://Wait 1 Step to reset the delay counter befor start to write
		iStateModbus_CP := iStateModbusRead;
		
			iStateModbusWrite := 1;
				iStateModbusRead := - 1;	
				
		//Timeout
		IF timTimeout.Q THEN
			iStateModbusError := 300;
		END_IF	

END_CASE


(*------------------------------------------------------------------------------------------State Machine Write---------------------------------------------------------------------------------------------*)	
	
CASE iStateModbusWrite OF	
	
	1://Write target Power for EHE and HB to the Honeywell controller
		iStateModbus_CP := iStateModbusWrite;	
		
		fbMBWrite_FC16.nQuantity := 7;
			fbMBWrite_FC16.nMBAddr := 0;
				fbMBWrite_FC16.bExecute := TRUE;
		
		//Write Data in the Sendbuffer
		arrBuffer_FC16[1] := BYTE_TO_WORD(byHBCounter);
			arrBuffer_FC16[2] := REAL_TO_WORD((rTargetPowerEHEH01_1 * 10));
		arrBuffer_FC16[3] := REAL_TO_WORD((rTargetPowerEHEH01_2 * 10)); 	
			arrBuffer_FC16[4] := REAL_TO_WORD((rTargetPowerEHEH01_3 * 10));
		arrBuffer_FC16[5] := REAL_TO_WORD((rTargetPowerEHEH08_1 * 10)); 
			arrBuffer_FC16[6] := REAL_TO_WORD((rTargetPowerEHEH08_2 * 10)); 	
		arrBuffer_FC16[7] := REAL_TO_WORD((rTargetPowerEHEH09_1 * 10));
	
		IF fbMBWrite_FC16.bBusy THEN timDelay.IN := TRUE; END_IF

		//Wait for Delay and then next step
		IF NOT fbMBWrite_FC16.bBusy AND NOT fbMBWrite_FC16.bError AND timDelay.Q THEN
			fbMBWrite_FC16.bExecute := FALSE;
				timDelay.IN := FALSE;
					bErrorFunction := FALSE; 
						//Restart from new with the Read out part
						iStateModbusRead := 1;
							iStateModbusWrite := 0;
		END_IF
				
		//Error or Timout
		IF FPError_FC_16.Q OR timTimeout.Q THEN
			iStateModbusError := 300;
		END_IF

END_CASE

(*------------------------------------------------------------------------------------------State Machine Error---------------------------------------------------------------------------------------------*)	

CASE iStateModbusError OF
	
	300://Error
		iStateModbus_CP := iStateModbusError;
			timDelay.IN := FALSE;
				fbMBRead_FC4.bExecute := FALSE;
					fbMBWrite_FC16.bExecute := FALSE;
						bErrorFunction := TRUE;	
							//Restart from new with the Read out part after an Error
							iStateModbusRead := 1;	
								iStateModbusError := 0;
									iStateModbusWrite := 0;
END_CASE

(*------------------------------------------------------------------------------------------Modbus TCP Functions---------------------------------------------------------------------------------------------*)

fbMBRead_FC4(sIPAddr:= sIPAdress, nUnitID := byUnitID, nTCPPort:= 12000, cbLength:= SIZEOF(arrBuffer_FC4), pDestAddr:= ADR(arrBuffer_FC4), tTimeout:= T#10S );
	FPError_FC_4(CLK:= fbMBRead_FC4.bError, Q=> );

fbMBWrite_FC16(sIPAddr:= sIPAdress, nTCPPort:= 12000, nUnitID := byUnitID, cbLength:= SIZEOF(arrBuffer_FC16), pSrcAddr:= ADR(arrBuffer_FC16), tTimeout:= T#10S );
	FPError_FC_16(CLK:= fbMBWrite_FC16.bError, Q=> );

END_FUNCTION_BLOCK

// ---- FBs/FB_CV_WORD_TO_DWORD.TcPOU
FUNCTION_BLOCK FB_CV_WORD_TO_DWORD
VAR_INPUT
	wInputValue_1				: WORD;								//Input value that is converted into the output value
	wInputValue_2				: WORD;								//Input value that is converted into the output value
	eByteOrderForConvert		: eByteOrder;						//Byte Format
END_VAR
VAR_OUTPUT
	dwOutputValue				: DWORD;							//Converted output value							
END_VAR
VAR
END_VAR

//Creator : Kai Ebensperger
//Company : Lynus AG
//Date : 28.04.2021
//Version : 1.0.0.0

//With this functionblock its possible to convert a certain Datatyp in a other Datatype
//The byte order can be selected between BigEndian and LittleEndian
//WORD TO DWORD
//Created for the Edge Device Lib over Modbus TCP
//Modbus TCP is WORD oriented

IF eByteOrderForConvert = eByteOrder.eBigEndian THEN
	dwOutputValue := SHL(WORD_TO_DWORD(wInputValue_1),16) + WORD_TO_DWORD(wInputValue_2);
ELSE
	dwOutputValue := SHL(WORD_TO_DWORD(wInputValue_2),16) + WORD_TO_DWORD(wInputValue_1);
END_IF

END_FUNCTION_BLOCK

// ---- POUs/prgPV.TcPOU
PROGRAM prgPV
VAR
	fbFroniusPV			: FB_Symo_PV_Inverter_INT_1_DM_30_Inverter;
	fbPV				: FB_PV_Power_Ext_Input;
	fbPVCounter			: FB_EnergyCounter;
	byErrorWarningPV	: BYTE;							//{#lynus.ag#()}
	lrPowerTotalPV		: LREAL;						//{#lynus.ag#()}
END_VAR
VAR PERSISTENT
	lrCounterPV			: LREAL;						//{#lynus.ag#()}
END_VAR

//Creator : Kai Ebensperger
//Company : Lynus AG
//Updated : M.Schwarzmann
//Date : 20.06.2022
//Version : 1.0.0.1

//changes
//1.0.0.1 : added fbPVCounter, changed lrCounterPV origin


//Unit Ids from each Inverter
fbFroniusPV.arrUnitID_Inverter[1] := 1;
fbFroniusPV.arrUnitID_Inverter[2] := 2;
fbFroniusPV.arrUnitID_Inverter[3] := 3;
fbFroniusPV.arrUnitID_Inverter[4] := 4;
fbFroniusPV.arrUnitID_Inverter[5] := 5;
fbFroniusPV.arrUnitID_Inverter[6] := 6;
fbFroniusPV.arrUnitID_Inverter[7] := 7;

fbFroniusPV(
	bEnable:= TRUE, 
	sIPAdress:= '10.68.10.80', 
	arrUnitID_Inverter:= , 
	arrDataSymo10=> , 
	stDataEMPower_PV=> , 
	stDataEMCounter_PV=> , 
	diNrOfEM_OUT_PV=> );

IF fbFroniusPV.stDataEMPower_PV.byErrorWarning <> 0 THEN fbPV.bExtErrorPv := TRUE; ELSE fbPV.bExtErrorPv := FALSE; END_IF
	
fbPV(
	bEnable:= TRUE, 
	bExtErrorPv:= , 
	lrExtPvPower:= fbFroniusPV.stDataEMPower_PV.lrPowerTotal, 
	lrExtTotalCounterEnergy_Consumption:= , 
	lrExtTotalCounterEnergy_Production:= fbFroniusPV.stDataEMCounter_PV.lrTotalCounterEnergy_Production, 
	lrExtCounterEnergyT1_Consumption:= , 
	lrExtCounterEnergyT2_Consumption:= , 
	lrExtCounterEnergyT1_Production:= , 
	lrExtCounterEnergyT2_Production:= , 
	stDataPv=> , 
	diNrOfPv_OUT=> );	
	
byErrorWarningPV := fbPV.stDataPv.byErrorWarning;
	lrPowerTotalPV := fbPV.stDataPv.lrPower;

fbPVCounter(
	byActiveTariff:= 1, 
	lrPowerInput:= 0 - lrPowerTotalPV, 
	lrTotalCounterEnergy_Consumption=> , 
	lrTotalCounterEnergy_Production=> , 
	lrCounterEnergyT1_Consumption=> , 
	lrCounterEnergyT2_Consumption=> , 
	lrCounterEnergyT1_Production=> , 
	lrCounterEnergyT2_Production=> );
	
IF fbPVCounter.lrTotalCounterEnergy_Production > lrCounterPV THEN  	
	lrCounterPV := fbPVCounter.lrTotalCounterEnergy_Production;
END_IF

END_PROGRAM

// ---- FBs/FB_EnergyCounter.TcPOU
FUNCTION_BLOCK FB_EnergyCounter
VAR_INPUT
	byActiveTariff						: BYTE;						//Active Tariff
	lrPowerInput						: LREAL;					//Input Power in kW
END_VAR
VAR_OUTPUT PERSISTENT
	lrTotalCounterEnergy_Consumption	: LREAL;					//Total Counter for Energy consumption with unit kWh
	lrTotalCounterEnergy_Production		: LREAL;					//Total Counter for Energy production with unit kWh
	lrCounterEnergyT1_Consumption		: LREAL;					//Total counter for energy Tariff 1 consumption with unit kWh
	lrCounterEnergyT2_Consumption		: LREAL;					//Total counter for energy Tariff 2 consumption with unit kWh
	lrCounterEnergyT1_Production		: LREAL;					//Total counter for energy Tariff 1 production with unit kWh
	lrCounterEnergyT2_Production		: LREAL;					//Total counter for energy Tariff 2 production with unit kWh
END_VAR
VAR
	TaskInfo							: GETCURTASKINDEX;			//Function to get the Task Index
	byWorkMode							: BYTE;						//Work Mode for calculation (1 = Production, 2 = Consumption)
	udiCycleTime						: UDINT;					//Cycle Time
	lrCyclesForSecond					: LREAL;					//Needed cycles for 1 Second
	uiCounterConsumption				: UINT;						//Counter for Cycles in Consumption Mode
	uiSecondsConsumption				: UINT;						//Elapses Seconds for Consumption
	rHourConsumption					: REAL;						//Elapsed Hours for Consumption
	uiCounterProduction					: UINT;						//Counter for Cycles in Production Mode
	uiSecondsProduction					: UINT;						//Elapses Seconds for Production
	rHourProduction						: REAL;						//Elapsed Hours for Production
	lrkW_Consumption_CP					: LREAL;					//Power to compare in Consumption Mode
	lrkW_Production_CP					: LREAL;					//Powet to compare in Production Mode
END_VAR

//Creator : Kai Ebensperger
//Company : Lynus AG
//Date : 16.11.2021
//Version : 1.0.0.0

//This function block can be used to count different Energy Counter
//Positive Values mens comsumption
//Negative Values means production 

(*--------------------------------------------------------------------------Limits-----------------------------------------------------------------------------------*)

byActiveTariff := LIMIT(1,byActiveTariff,2);

(*---------------------------------------------------------------------------Logic-----------------------------------------------------------------------------------*)

//Get Task Index
TaskInfo(index=> );
	//Cycle Time in ms
	IF TwinCAT_SystemInfoVarList._TaskInfo[TaskInfo.index].CycleTime <> 0 THEN
		udiCycleTime := TwinCAT_SystemInfoVarList._TaskInfo[TaskInfo.index].CycleTime / 10000;
	END_IF

//Cycles for 1 Second
IF udiCycleTime > 0 THEN 
	lrCyclesForSecond := (1 / UDINT_TO_LREAL(udiCycleTime)) * 1000; 
END_IF

IF lrCyclesForSecond <> 0 THEN

	uiCounterConsumption := uiCounterConsumption + 1;
		uiCounterProduction := uiCounterProduction + 1;
	
	//Calculate the Time	
	IF uiCounterProduction >= lrCyclesForSecond THEN uiSecondsProduction := uiSecondsProduction + 1; uiCounterProduction := 0; END_IF
		rHourProduction := UINT_TO_REAL(uiSecondsProduction) / 3600;
	IF uiCounterConsumption >= lrCyclesForSecond THEN uiSecondsConsumption := uiSecondsConsumption + 1; uiCounterConsumption := 0; END_IF
		rHourConsumption := UINT_TO_REAL(uiSecondsConsumption) / 3600;
	
	//Production
	IF lrkW_Production_CP <> lrPowerInput THEN
		IF byWorkMode = 1 THEN 
			//Production Tariff 1
			IF byActiveTariff = 1 THEN 
				lrCounterEnergyT1_Production := lrCounterEnergyT1_Production + ((lrkW_Production_CP * - 1) * rHourProduction); 
					lrkW_Production_CP := lrPowerInput;
			END_IF
			//Production Tariff 2
			IF byActiveTariff = 2 THEN 
				lrCounterEnergyT2_Production := lrCounterEnergyT2_Production + ((lrkW_Production_CP * - 1) * rHourProduction); 
					lrkW_Production_CP := lrPowerInput;
			END_IF
		ELSE
			lrkW_Production_CP := 0;
		END_IF
				rHourProduction := 0; uiSecondsProduction := 0;  uiCounterProduction := 0;	
	END_IF
	
	//Consumption
	IF lrkW_Consumption_CP <> lrPowerInput THEN
		IF byWorkMode = 2 THEN  
			//Consumption Tariff 1
			IF byActiveTariff = 1 THEN 
				lrCounterEnergyT1_Consumption := lrCounterEnergyT1_Consumption + (lrkW_Consumption_CP * rHourConsumption); 
					lrkW_Consumption_CP := lrPowerInput;
			END_IF
			//Consumption Tariff 2
			IF byActiveTariff = 2 THEN 
				lrCounterEnergyT2_Consumption := lrCounterEnergyT2_Consumption + (lrkW_Consumption_CP * rHourConsumption); 
					lrkW_Consumption_CP := lrPowerInput;
			END_IF
		ELSE
			lrkW_Consumption_CP := 0;
		END_IF
				rHourConsumption := 0; uiSecondsConsumption := 0;  uiCounterConsumption := 0;	
	END_IF

END_IF

//Total Consumption and Production
lrTotalCounterEnergy_Consumption := lrCounterEnergyT1_Consumption + lrCounterEnergyT2_Consumption;
	lrTotalCounterEnergy_Production := lrCounterEnergyT1_Production + lrCounterEnergyT2_Production;

//Switch between the Work modes
IF lrPowerInput <= 0 THEN byWorkMode := 1; ELSE byWorkMode := 2; END_IF

END_FUNCTION_BLOCK

// ---- POUs/prgXelect.TcPOU
PROGRAM prgXelect
VAR
	fbBatt					: FB_Xelectrix_Powerbox;			//{#lynus.ag#()}
	fbCounter				: FB_EnergyCounter;
	byErrorWarningBattery	: BYTE;								//{#lynus.ag#()}
	lrBattGridPower			: LREAL;							//{#lynus.ag#()}
END_VAR
VAR PERSISTENT
	lrkWh_Charge			: LREAL;							//{#lynus.ag#()}
	lrkWh_Discharge			: LREAL;							//{#lynus.ag#()}
END_VAR

fbBatt(
	bEnable:= , 
	bActivateControl:= TRUE, 
	byUnitID:= 1, 
	byPriority:= , 
	diNrOfEMS_IN:= prgEMS.EMS.diNrOfEMS_OUT, 
	lrMaxCapacityBattery:= 240, 
	sIPAdress:= '10.68.11.30', 
	bReset:= , 
	stDataXelectrix=> , 
	stDataBatt=> , 
	stDataBattInverter=> , 
	stDataEMPower_Grid=> , 
	stDataEMCounter_Grid=> , 
	diNrOfBatt_OUT=> , 
	diNrOfBattInverter_OUT=> , 
	diNrOfEM_OUT_Grid=> , 
	lrMaxCapacityBattery_OUT=> );
	
byErrorWarningBattery := fbBatt.stDataBatt.byErrorWarning;	

fbCounter(
	byActiveTariff:= 1, 
	lrPowerInput:= fbBatt.stDataBatt.lrPower, 
	lrTotalCounterEnergy_Consumption=> , 
	lrTotalCounterEnergy_Production=> , 
	lrCounterEnergyT1_Consumption=> , 
	lrCounterEnergyT2_Consumption=> , 
	lrCounterEnergyT1_Production=> , 
	lrCounterEnergyT2_Production=> );

IF fbCounter.lrTotalCounterEnergy_Consumption > lrkWh_Discharge THEN
	lrkWh_Discharge := fbCounter.lrTotalCounterEnergy_Consumption;
END_IF
	IF fbCounter.lrTotalCounterEnergy_Production > lrkWh_Charge THEN
		lrkWh_Charge := fbCounter.lrTotalCounterEnergy_Production;
	END_IF

END_PROGRAM

// ---- POUs/prgPerData.TcPOU
PROGRAM prgPerData
VAR
	fbPerData			: FB_WritePersistentData_CX81xx;
END_VAR

fbPerData(
	eSaveModeData:= eUSVSaveMode.eSaveWhenPowerfail, 
	bLoadPersistentDataOk=> , 
	bPowerFailDetect=> , 
	bError=> , 
	bySaveProcess=> , 
	dwStorageLast24h=> , 
	udiErrorCode=> );

END_PROGRAM

// ---- POUs/prgHouse.TcPOU
PROGRAM prgHouse
VAR
	fbHouse					: FB_HouseC_Power_Virtual;
	fbHouse2				: FB_HouseC_Power_Virtual_v2;
	lrPowerHouse			: LREAL;	//{#lynus.ag#()}
	lrPowerHouse2			: LREAL;
	bStateEnabelHouse		: BOOL;		//{#lynus.ag#()}
	lrPowerHouseReal		: LREAL;	//{#lynus.ag#()}
	lrPowerHouseReal2		: LREAL;
	bStateEnableRaceStable	: BOOL;		//{#lynus.ag#()}
	lrPowerRaceStable		: LREAL;	//{#lynus.ag#()}
END_VAR
VAR PERSISTENT
	bEnableHouse		: BOOL;		//{#lynus.ag#()}
	bEnableHouse2		: BOOL;
	bEnableRaceStable	: BOOL;		//{#lynus.ag#()}
	lrCounterHouse		: LREAL;	//{#lynus.ag#()}
END_VAR

//Creator : Kai Ebensperger
//Company : Lynus AG
//Updated : M.Schwarzmann
//Date : 29.04.2022
//Version : 1.0.0.1

//changes
//1.0.0.1 : added lrPowerHouseReal Variable, which subtracts the received Power of Electricity Meter from the calculated virtual House Power; added EMS Part for Power Consumption Race Stable

// -- TestBegin
fbHouse2(bEnable:= bEnableHouse2, diNrOfEMS_IN:= prgEMS.EMS.diNrOfEMS_OUT, stDataHouseC=> , diNrOfHouseC_OUT=> );
	lrPowerHouse2 := fbHouse2.stDataHouseC.lrPower;
	
IF (lrPowerHouse2 - prgHoneywell.dwElectricMeterPower) >= 0 THEN
	lrPowerHouseReal2 := lrPowerHouse2 - prgHoneywell.dwElectricMeterPower;
ELSE
	lrPowerHouseReal2 := 0;
END_IF

// -- TestEnd

fbHouse(bEnable:= bEnableHouse, diNrOfEMS_IN:= prgEMS.EMS.diNrOfEMS_OUT, stDataHouseC=> , diNrOfHouseC_OUT=> );
	lrPowerHouse := fbHouse.stDataHouseC.lrPower;
		bStateEnabelHouse := fbHouse.stDataHouseC.bEnabled;

IF (lrPowerHouse - prgHoneywell.dwElectricMeterPower) >= 0 THEN
	lrPowerHouseReal := lrPowerHouse - prgHoneywell.dwElectricMeterPower;
ELSE
	lrPowerHouseReal := 0;
END_IF

IF fbHouse.stDataHouseC.lrTotalCounterEnergy_Consumption > lrCounterHouse THEN
	lrCounterHouse := fbHouse.stDataHouseC.lrTotalCounterEnergy_Consumption;
END_IF

//EMS Part for Power Consumption Race Stable

IF bEnableRaceStable THEN
    bStateEnableRaceStable := TRUE;
    lrPowerRaceStable := prgHoneywell.dwElectricMeterPower;
ELSE
	bStateEnableRaceStable := FALSE;
	lrPowerRaceStable := 0;
END_IF

END_PROGRAM

// ---- FBs/FB_HouseC_Power_Virtual_v2.TcPOU
FUNCTION_BLOCK FB_HouseC_Power_Virtual_v2
VAR_INPUT PERSISTENT
	bEnable									: BOOL;													//{#lynus.ag#()} //Enable the Fuctionblock and his logic
	diNrOfEMS_IN							: DINT;													//Number of EMS from what this Device received Data
END_VAR
VAR_INPUT
	bSetDefault								: BOOL;													//With this Input can set the default Value from the Counter from the Input to the Counter at the Output									
	lrCounterConsumptionSetDefault			: LREAL;												//Set Default value for Consumption Counter
	lrCounterProductionSetDefault			: LREAL;												//Set Default value for Production Counter
END_VAR
VAR_OUTPUT
	stDataHouseC							: ST_HouseConsumption_Output;							//{#lynus.ag#()} //House consumption output data
	diNrOfHouseC_OUT						: DINT;													//Active Number from the House connection for using on other functions
END_VAR
VAR
	{attribute 'hide'}
	fbHouseC								: FB_HouseConsumption;									//Function for House consumption
	{attribute 'hide'}
	fbNumberDevice							: FB_NumberOfDevice;									//Function block to calcualte the number of the Device
	{attribute 'hide'}
	TaskIndex								: GETCURTASKINDEX;										//Function to read out the task index	
	{attribute 'hide'}
	timSaveCSProd							: TON;													//Timer to save the Counter Status from production on persistent data
	{attribute 'hide'}
	timSaveCSCons							: TON;													//Timer to save the Counter Status from Consumption on persistent data
	{attribute 'hide'}
	timDissableFunctions					: TON;													//Timer to dissable the Function after Lynus_Standards.Constants_General.tTimeDissableLynusFunctions Days without connection to the Lynus Cloud
	{attribute 'hide'}
	timResetConnectionOnGVL					: TON;													//Timer to try reset the connection Flag on the GVL. (When somebody delete the Connection Function and make only a onlinechange)
	{attribute 'hide'}
	FPSetDefault							: R_TRIG;												//Internal positive Edge
	{attribute 'hide'}
	arrPD									: ARRAY[1..4] OF FB_PersistentData_Number;				//Function to save persistent data 
	{attribute 'hide'}
	bError									: BOOL;													//Error from external Devices
	{attribute 'hide'}
	byWaitInStep							: BYTE;													//Wait in Step before start to clean data on PLC
	{attribute 'hide'}
	iStateGVLData							: INT;													//State machine to handle the data on the GVL
	{attribute 'hide'}
	diCounterForGVL							: DINT;													//Counter to clean old data on GVL
	{attribute 'hide'}
	udicycleTime							: UDINT;												//Cycletime of plc
	{attribute 'hide'}
	lrPowerProduction						: LREAL;												//Complete Power Production from al Devices of this EMS in kW 
	{attribute 'hide'}
	lrPowerBattery							: LREAL;												//Complete Battery Power from al Batterys of this EMS in kW 
	{attribute 'hide'}
	lrPowerGrid								: LREAL;												//Complete Grid Power from al Grids of this EMS in kW 
	{attribute 'hide'}
	lrCounterConsumption_CP					: LREAL;												//Counter Status Consumption with Unit kW/h to compare for save persistent
	{attribute 'hide'}
	lrCounterProduction_CP					: LREAL;												//Counter Status Production with Unit kW/h to compare for save persistent
	{attribute 'hide'}
	lrTotalPower							: LREAL;												//Total power with unit kW
	{attribute 'hide'}
	lrTotalPower_CP							: LREAL;												//Total power with unit kW to trigger the calculation for energy
	{attribute 'hide'}
	lrCyclesForMinute						: LREAL;												//Cycles what the plc need for 1 minute 
	{attribute 'hide'}
	lrPastTime								: LREAL;												//Past time in hours 
	{attribute 'hide'}
	lrSumToCalculate						: LREAL;												//Actual sum of the energy counters before start the calculation with unit kW/h
	{attribute 'hide'}
	liLPPower								: LINT;													//Loop to calculate the total power
END_VAR
VAR PERSISTENT
	{attribute 'conditionalshow'}
	lrCounterConsumption					: LREAL;												//Counter Status Consumption with Unit kW/h
	{attribute 'conditionalshow'}
	lrCounterProduction						: LREAL;												//Counter Status Production with Unit kW/h
END_VAR

//Creator : Kai Ebensperger
//Company : Lynus AG
//Date : 15.06.2021
//Version : 1.0.0.0

//With this function block its possible to show the power data from a house.
//The power data in this function block is calculated by all the other consumers and producers. So the output data is not messured.
//Use only one of this Function block per each EMS
//NOTE : The output from this Function Block is not 100% perfect why the value is only calculatet and not messured.

//NOTE for diNr.....Designation => 
//_IN = Here Data come in from other Functions or go out to other functions about the GVL
//_OUT = Here Data go out to other functions about the GVL

(*------------------------------------------------------------Limits----------------------------------------------------------------------------------*)

diNrOfEMS_IN := LIMIT(0,diNrOfEMS_IN,Constants_Energy.diMaxNumberOfEMS);

(*-------------------------------------------------------------Calcualte the number of House Consumption---------------------------------------------------------------*)

fbNumberDevice(
	diActualNumberOfDevices:= Lynus_Standards.GVL_Energy.stNumberOfDevices.diNumberOfHouseConsumption, 
	diMaxNumberOfDevices:= Constants_Energy.diMaxNumberOfHouseConsumptions, 
	udiCounterOnlineChange:= TwinCAT_SystemInfoVarList._AppInfo.OnlineChangeCnt, 
	bNumberIsCalculatet=> , 
	bFPNumberIsCalculatet=> , 
	bOnlineChange=> , 
	diNumberForThisDevice=> diNrOfHouseC_OUT, 
	diNumberOfTotalDevices=> );

//Write new Numer on GVL
IF fbNumberDevice.bFPNumberIsCalculatet THEN
	Lynus_Standards.GVL_Energy.stNumberOfDevices.diNumberOfHouseConsumption := fbNumberDevice.diNumberOfTotalDevices;	
END_IF 

//Delete old Number on GVL
IF fbNumberDevice.bOnlineChange THEN 
	Lynus_Standards.GVL_Energy.stNumberOfDevices.diNumberOfHouseConsumption := diNrOfHouseC_OUT;	
		iStateGVLData := 1; 
END_IF

(*-------------------------------------------------------------Calcualte the power of the house---------------------------------------------------------------*)	

lrPowerProduction := 0;
	lrPowerBattery := 0;
		lrPowerGrid := 0;
			bError := FALSE;

//Batterypower
FOR liLPPower := 1 TO Constants_Energy.diMaxNumberOfBatterys BY 1 DO
	lrPowerBattery := lrPowerBattery + Lynus_Standards.GVL_Energy.stDataOfBatterys[diNrOfEMS_IN,liLPPower].lrPower;	
		IF Lynus_Standards.GVL_Energy.stDataOfBatterys[diNrOfEMS_IN,liLPPower].byErrorWarning = 2 THEN bError := TRUE; END_IF 
END_FOR 
 	//Generator power
	FOR liLPPower := 1 TO Constants_Energy.diMaxNumberOfGenerators BY 1 DO
		lrPowerProduction := lrPowerProduction + Lynus_Standards.GVL_Energy.stDataOfGenerators[liLPPower].lrPowerProduction;	
			IF Lynus_Standards.GVL_Energy.stDataOfGenerators[liLPPower].byErrorWarning = 2 THEN bError := TRUE; END_IF		
	END_FOR 
		//PV power
		FOR liLPPower := 1 TO Constants_Energy.diMaxNumberOfPvSystems BY 1 DO
			lrPowerProduction := lrPowerProduction + Lynus_Standards.GVL_Energy.stDataOfPvSystems[liLPPower].lrPowerProduction;	
				IF Lynus_Standards.GVL_Energy.stDataOfPvSystems[liLPPower].byErrorWarning = 2 THEN bError := TRUE; END_IF		
		END_FOR	
			//Grid power	
			FOR liLPPower := 1 TO Constants_Energy.diMaxNumberOfGridConnections BY 1 DO
				lrPowerGrid := lrPowerGrid + Lynus_Standards.GVL_Energy.stDataGridConnections[diNrOfEMS_IN,liLPPower].lrPower;	
					IF Lynus_Standards.GVL_Energy.stDataGridConnections[diNrOfEMS_IN,liLPPower].byErrorWarning = 2 THEN bError := TRUE; END_IF 
			END_FOR 

//Complete power
lrTotalPower := lrPowerProduction + lrPowerGrid + lrPowerBattery;
	lrTotalPower := LIMIT(0,lrTotalPower,100000);							

(*-------------------------------------------------------------Calcualte the energy of the house---------------------------------------------------------------*)
							
//Read out the Taskindex
TaskIndex(index=> );							

//Set default Value
FPSetDefault(CLK:= bSetDefault, Q=> );
	IF FPSetDefault.Q THEN 
		lrCounterConsumption_CP := lrCounterConsumptionSetDefault;
			lrCounterProduction_CP := lrCounterProductionSetDefault;
	END_IF
						
//Save the persistent counter status to the counter status for compare on the first plc cycle	
IF TwinCAT_SystemInfoVarList._TaskInfo[TaskIndex.index].FirstCycle THEN 
	lrCounterConsumption_CP := lrCounterConsumption;
		lrCounterProduction_CP := lrCounterProduction;
END_IF											

//Timer to save the Energy Counters persistent every 12 hours											
timSaveCSProd(IN:= lrCounterProduction <> lrCounterProduction_CP, PT:= T#12H, Q=> , ET=> );
	timSaveCSCons(IN:= lrCounterConsumption <> lrCounterConsumption_CP, PT:= T#12H, Q=> , ET=> );

IF timSaveCSProd.Q THEN lrCounterProduction := lrCounterProduction_CP; END_IF 
	IF timSaveCSCons.Q THEN lrCounterConsumption := lrCounterConsumption_CP; END_IF  
	
//Write Data when the Event Based saving on persitent Data is not active
IF NOT arrPD[3].bEventBasedActive AND NOT arrPD[4].bEventBasedActive THEN
	lrCounterProduction := lrCounterProduction_CP;
		lrCounterConsumption := lrCounterConsumption_CP;
END_IF   
			
//Read out the cycle time to calculate the energy counters
//Cycle Time in MS
udicycleTime := TwinCAT_SystemInfoVarList._TaskInfo[TaskIndex.index].CycleTime / 10000;

//Calculate the cycles what is needed for 1 Minute
lrCyclesForMinute := UDINT_TO_LREAL((1 * udicycleTime)) / 60000;	

//Calculate past time in hours
lrPastTime := lrPastTime + (lrCyclesForMinute / 60);

//Calculate the Energy when the power data change and start then from new
IF MEMCMP(ADR(lrTotalPower),ADR(lrTotalPower_CP),SIZEOF(lrTotalPower_CP)) <> 0 THEN
	//INFO : Negative Value at the moment is not in use about the limitation of the Total power
	IF lrSumToCalculate < 0 THEN
		lrCounterProduction_CP := lrCounterProduction_CP + (lrSumToCalculate * - 1);
	ELSE
		lrCounterConsumption_CP := lrCounterConsumption_CP + lrSumToCalculate;
	END_IF
		lrSumToCalculate := 0;
			lrPastTime := 0;
				lrTotalPower_CP := lrTotalPower;
END_IF

//Calculate the sum after the calculation why we must calculate after the power change
lrSumToCalculate := lrTotalPower * lrPastTime;

(*-------------------------------------------------------------Service from Backend is ready and check the connection to backen for dissabel/enable Function---------------------------------------------------------------*)

//Try to reset the variable for connection on the GVL. When all is normal then the Lynus Mqtt connection function set this variable to true in the next cycle
//When we have no connection to the backend then after Lynus_Standards.Constants_General.tTimeDissableLynusFunctions days the Function is dissabled with all of his functionalities
timResetConnectionOnGVL(IN:= NOT timResetConnectionOnGVL.Q, PT:= T#1H, Q=> , ET=> );
	IF timResetConnectionOnGVL.Q THEN Lynus_Standards.GVL_Communicator.bStateConnectionToEnableFunctions := FALSE; END_IF
		IF NOT Lynus_Standards.GVL_Communicator.bStateConnectionToEnableFunctions THEN timDissableFunctions.IN := TRUE; ELSE timDissableFunctions.IN := FALSE; END_IF  
			timDissableFunctions(IN:= , PT:= Lynus_Standards.Constants_General.tTimeDissableLynusFunctions, Q=> , ET=> );

(*-----------------------------------------------------------------------------Error ----------------------------------------------------------------------------*)

IF timDissableFunctions.Q THEN fbHouseC.bWarning := TRUE; fbHouseC.iWarningCode := 0; ELSE fbHouseC.bWarning := FALSE; END_IF 	
	IF Lynus_Standards.GVL_Energy.stNumberOfDevices.diNumberOfHouseConsumption > Constants_Energy.diMaxNumberOfHouseConsumptions OR bError THEN fbHouseC.bError := TRUE; ELSE fbHouseC.bError := FALSE; END_IF 
		IF Lynus_Standards.GVL_Energy.stNumberOfDevices.diNumberOfHouseConsumption > Constants_Energy.diMaxNumberOfHouseConsumptions THEN fbHouseC.iErrorCode := 1;
		ELSIF bError THEN fbHouseC.iErrorCode := 0; 
		END_IF  

(*------------------------------------------------------------------FB House----------------------------------------------------------------------------*)	
	
fbHouseC(
	bEnable:= bEnable AND NOT timDissableFunctions.Q,
	bError:= , 
	bWriteWithDelay:= TRUE, 
	iErrorCode:= , 
	iWarningCode:= , 
	lrTotalCounterEnergy_Consumption:= lrCounterConsumption_CP * 1000, 
	lrTotalCounterEnergy_Production:= lrCounterProduction_CP * 1000, 
	lrCounterEnergyT1_Consumption:= lrCounterConsumption_CP * 1000, 
	lrCounterEnergyT2_Consumption:= , 
	lrCounterEnergyT1_Production:= lrCounterProduction_CP * 1000, 
	lrCounterEnergyT2_Production:= , 
	lrPowerHouseConsumption:= lrTotalPower * 1000, 
	tTimDelayOutput:= T#5S, 
	stDataHouseCOut=> , 
	stDataHouseCOutDelay=> stDataHouseC);
	
	(*-----------------------------------------------------------Handle data to Global structure for the House consumption-----------------------------------------------------------------*)

CASE iStateGVLData OF
	
	0://Init Step
		byWaitInStep := 0;
			diCounterForGVL := 1;
	
	1://Wait for 4 Steps before clean al Data on GVL
		byWaitInStep := byWaitInStep + 1;
			IF byWaitInStep >= 4 AND fbNumberDevice.bNumberIsCalculatet THEN iStateGVLData := 2; END_IF
				//To much Devices, back to the Init step
				IF byWaitInStep >= 4 AND NOT fbNumberDevice.bNumberIsCalculatet THEN iStateGVLData := 0; END_IF	
			
	2://Clear all Data in GVL
		Lynus_Standards.GVL_Energy.stDataHouseConsumptions[diCounterForGVL].bEnabled := FALSE;
			Lynus_Standards.GVL_Energy.stDataHouseConsumptions[diCounterForGVL].byErrorWarning := 0;
				Lynus_Standards.GVL_Energy.stDataHouseConsumptions[diCounterForGVL].lrPowerConsumption := 0;
					Lynus_Standards.GVL_Energy.stDataHouseConsumptions[diCounterForGVL].lrPower := 0;
						Lynus_Standards.GVL_Energy.stDataHouseConsumptions[diCounterForGVL].lrPowerProduction := 0;
		
		diCounterForGVL := diCounterForGVL + 1;
			diCounterForGVL := LIMIT(0,diCounterForGVL,Constants_Energy.diMaxNumberOfHouseConsumptions);
				//Back to the init step
				IF diCounterForGVL >= Constants_Energy.diMaxNumberOfHouseConsumptions THEN iStateGVLData := 0; END_IF
				
END_CASE 	 

IF diNrOfHouseC_OUT > 0 AND fbNumberDevice.bNumberIsCalculatet THEN
	Lynus_Standards.GVL_Energy.stDataHouseConsumptions[diNrOfHouseC_OUT].bEnabled := fbHouseC.stDataHouseCOut.bEnabled;
		Lynus_Standards.GVL_Energy.stDataHouseConsumptions[diNrOfHouseC_OUT].byErrorWarning := fbHouseC.stDataHouseCOut.byErrorWarning;
			Lynus_Standards.GVL_Energy.stDataHouseConsumptions[diNrOfHouseC_OUT].lrPowerConsumption := fbHouseC.stDataHouseCOut.lrPowerConsumption;
				Lynus_Standards.GVL_Energy.stDataHouseConsumptions[diNrOfHouseC_OUT].lrPower := fbHouseC.stDataHouseCOut.lrPower;
					Lynus_Standards.GVL_Energy.stDataHouseConsumptions[diNrOfHouseC_OUT].lrPowerProduction := fbHouseC.stDataHouseCOut.lrPowerProduction;
END_IF 	

(*----------------------------------------------------------Save persistent data----------------------------------------------------------------*)

arrPD[1](lrValue:= BOOL_TO_LREAL(bEnable), bEventBasedActive=> );
arrPD[2](lrValue:= DINT_TO_LREAL(diNrOfEMS_IN), bEventBasedActive=> );
arrPD[3](lrValue:= lrCounterConsumption, bEventBasedActive=> );
arrPD[4](lrValue:= lrCounterProduction, bEventBasedActive=> );

END_FUNCTION_BLOCK

// ---- POUs/prgGrid.TcPOU
PROGRAM prgGrid
VAR
	fbGrid					: FB_Grid_Power;
	fbCounter				: FB_EnergyCounter;
	lrGridPower				: LREAL;	//{#lynus.ag#()}
	byErrorWarningGrid		: BYTE;		//{#lynus.ag#()}
END_VAR
VAR PERSISTENT
	rSizeGrid				: REAL;		//{#lynus.ag#()}
	lrCounterGridCons		: LREAL;	//{#lynus.ag#()}
	lrCounterGridProd		: LREAL;	//{#lynus.ag#()}
END_VAR

fbGrid(
	bEnable:= TRUE, 
	diNrOfEMS_IN:= prgEMS.EMS.diNrOfEMS_OUT, 
	diNrOfEM_IN_Grid:= prgXelect.fbBatt.diNrOfEM_OUT_Grid, 
	rSizeGridConn:= rSizeGrid, 
	stDataGrid=> , 
	diNrOfGrid_OUT=> );
	
lrGridPower := fbGrid.stDataGrid.lrPower;
byErrorWarningGrid := fbGrid.stDataGrid.byErrorWarning;

fbCounter(
	byActiveTariff:= 1, 
	lrPowerInput:= lrGridPower, 
	lrTotalCounterEnergy_Consumption=> , 
	lrTotalCounterEnergy_Production=> , 
	lrCounterEnergyT1_Consumption=> , 
	lrCounterEnergyT2_Consumption=> , 
	lrCounterEnergyT1_Production=> , 
	lrCounterEnergyT2_Production=> );

IF fbCounter.lrTotalCounterEnergy_Consumption > lrCounterGridCons THEN
	lrCounterGridCons := fbCounter.lrTotalCounterEnergy_Consumption;
END_IF
	IF fbCounter.lrTotalCounterEnergy_Production > lrCounterGridProd THEN
		lrCounterGridProd := fbCounter.lrTotalCounterEnergy_Production;
	END_IF

END_PROGRAM

// ---- POUs/prgComLynus.TcPOU
PROGRAM prgComLynus
VAR
	fbCom			: FB_MqttCommunicator;
END_VAR

fbCom(
	bConnect:= TRUE, 
	sUserName:= 'b70e88c8-0481-4d36-92fe-45daf83d392d', 
	sUserPassword:= '31c9e512-5d63-471e-8e0c-6ecec0b71d43', 
	eSavePositionCertificate:= eSavePositionOnPLC.ePostionHardDisk, 
	bConnected=> , 
	bError=> , 
	hrErrorCode=> , 
	eConnectionState=> , 
	eErrorMessage_Out=> );

END_PROGRAM
